// TIA Portal V15.1 export
// export: Created 2024-06-21T08:41:25.4173155Z, ExportSetting WithDefaults, DisplayName Totally Integrated Automation Portal, DisplayVersion V15.1 Update 5, DisplayName TIA Portal Openness, DisplayVersion V15.1 Update 5, DisplayName SINAMICS Startdrive Advanced, DisplayVersion V15.1, DisplayName G130, G150, S120, S150, SINAMICS MV, S210, DisplayVersion V15.1, DisplayName G110M, G120, G120C, G120D, G120P, DisplayVersion V15.1, DisplayName STEP 7 Professional, DisplayVersion V15.1 Update 5, DisplayName STEP 7 Safety, DisplayVersion V15.1, DisplayName WinCC Professional, DisplayVersion V15.1 Update 5, DisplayName SIMATIC Visualization Architect, DisplayVersion V15.1
FUNCTION "209000NCP01Alarm" : Void   // FC258, FBD
TITLE = Alarm / 209000NCP01Alarm
{ S7_Optimized_Access := 'TRUE' }
AUTHOR : VCC
VERSION : 0.0.0.0
// =============================================================================
// This Module Controls All Alarm Sending To VD 
// =============================================================================
// stored: AutoNumber false, IsIECCheckEnabled false, SetENOAutomatically False, UDAEnableTagReadback false
BEGIN

REGION Network 1: **** 7.1 - Submodule - NonMachine **** Alarm Handler
   // Alarm Handler Send Requests
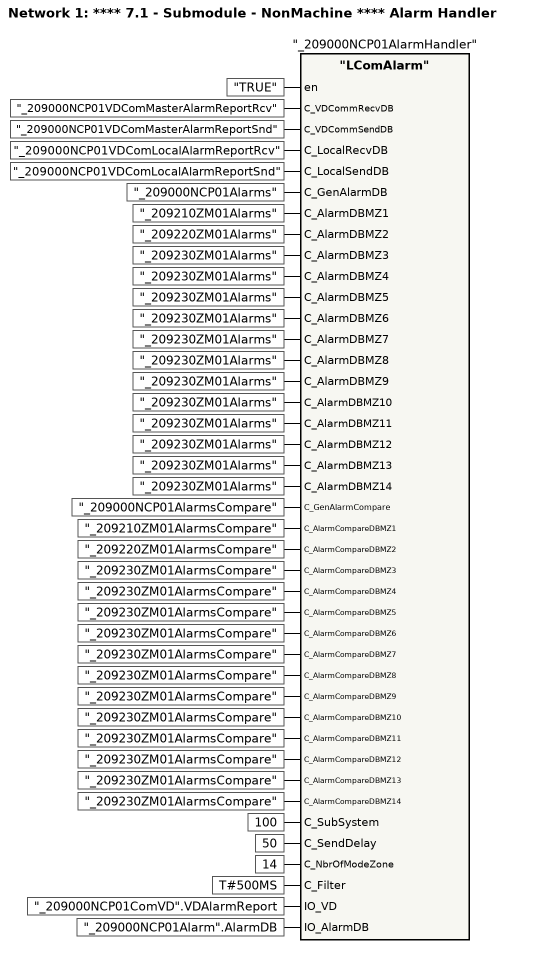
   IF "TRUE" THEN
       "_209000NCP01AlarmHandler"(C_VDCommRecvDB := "_209000NCP01VDComMasterAlarmReportRcv",   // "LComAlarm"
                               C_VDCommSendDB := "_209000NCP01VDComMasterAlarmReportSnd",
                               C_LocalRecvDB := "_209000NCP01VDComLocalAlarmReportRcv",
                               C_LocalSendDB := "_209000NCP01VDComLocalAlarmReportSnd",
                               C_GenAlarmDB := "_209000NCP01Alarms",
                               C_AlarmDBMZ1 := "_209210ZM01Alarms",
                               C_AlarmDBMZ2 := "_209220ZM01Alarms",
                               C_AlarmDBMZ3 := "_209230ZM01Alarms",
                               C_AlarmDBMZ4 := "_209230ZM01Alarms",
                               C_AlarmDBMZ5 := "_209230ZM01Alarms",
                               C_AlarmDBMZ6 := "_209230ZM01Alarms",
                               C_AlarmDBMZ7 := "_209230ZM01Alarms",
                               C_AlarmDBMZ8 := "_209230ZM01Alarms",
                               C_AlarmDBMZ9 := "_209230ZM01Alarms",
                               C_AlarmDBMZ10 := "_209230ZM01Alarms",
                               C_AlarmDBMZ11 := "_209230ZM01Alarms",
                               C_AlarmDBMZ12 := "_209230ZM01Alarms",
                               C_AlarmDBMZ13 := "_209230ZM01Alarms",
                               C_AlarmDBMZ14 := "_209230ZM01Alarms",
                               C_GenAlarmCompare := "_209000NCP01AlarmsCompare",
                               C_AlarmCompareDBMZ1 := "_209210ZM01AlarmsCompare",
                               C_AlarmCompareDBMZ2 := "_209220ZM01AlarmsCompare",
                               C_AlarmCompareDBMZ3 := "_209230ZM01AlarmsCompare",
                               C_AlarmCompareDBMZ4 := "_209230ZM01AlarmsCompare",
                               C_AlarmCompareDBMZ5 := "_209230ZM01AlarmsCompare",
                               C_AlarmCompareDBMZ6 := "_209230ZM01AlarmsCompare",
                               C_AlarmCompareDBMZ7 := "_209230ZM01AlarmsCompare",
                               C_AlarmCompareDBMZ8 := "_209230ZM01AlarmsCompare",
                               C_AlarmCompareDBMZ9 := "_209230ZM01AlarmsCompare",
                               C_AlarmCompareDBMZ10 := "_209230ZM01AlarmsCompare",
                               C_AlarmCompareDBMZ11 := "_209230ZM01AlarmsCompare",
                               C_AlarmCompareDBMZ12 := "_209230ZM01AlarmsCompare",
                               C_AlarmCompareDBMZ13 := "_209230ZM01AlarmsCompare",
                               C_AlarmCompareDBMZ14 := "_209230ZM01AlarmsCompare",
                               C_SubSystem := 100,
                               C_SendDelay := 50,
                               C_NbrOfModeZone := 14,
                               C_Filter := T#500MS,
                               IO_VD := "_209000NCP01ComVD".VDAlarmReport,
                               IO_AlarmDB := "_209000NCP01Alarm".AlarmDB);
   END_IF;
END_REGION
END_FUNCTION
